{attribute 'GeneratedUsingTerminal: EJ2521-0224-0016'}
{attribute addProperty BoxType "EJ2521-0224-0016"}
{attribute addProperty Id "ControlAT %Q*Control_DAEE1D523Frequency_valueAT %Q*UINT2"}
{attribute addProperty CRC "2458384612"}
{attribute addProperty Size "5"}
TYPE PTO_Control_9287F8E4 :
STRUCT
	{attribute addProperty Name "Control"}
	Control AT %Q* : Control_DAEE1D52;
	{attribute addProperty Name "Frequency_value"}
	Frequency_value AT %Q* : UINT;
END_STRUCT
END_TYPE

(* stored: Version 1.2.0.0, ProductVersion 3.1.4024.9
   DUT PTO_Control_9287F8E4: Id {78e795a3-61da-4253-abf8-07b5d2f0ba51} *)
